{attribute 'qualified_only'}
{attribute 'strict'}
TYPE VertexSmoothingSubType :
(
	NONE := 0, // Probably should check this is correct!
	CONSTANT_TOLERANCE_RADIUS := 1,
	DISTANCE_BETWEEN_INTERSETION_AND_VERTEX := 2,
	ADAPTIVE_TOLERANCE_RADIUS := 3
) UDINT;
END_TYPE

(* stored: Version 1.1.0.1, ProductVersion 3.1.4024.12
   DUT VertexSmoothingSubType: Id {082b0b68-eba1-4e07-ac18-c95ddbc3ae3e} *)
